PROGRAM Basic
VAR
	State:INT:= 0;
END_VAR

MC.Exec_Stop:= FALSE;
MC.Exec_Velocity := FALSE;

CASE state OF
	0:  MC.Exec_Stop:= TRUE;
		IF HMI.Bt_StartCycle THEN
			State:=1;
			MC.TargetDirection:= MC_Direction.MC_Positive_Direction;
			MC.TargetVel:= HMI.Tb_Vel;
		END_IF
	1:  MC.Exec_Velocity:=TRUE;
		IF HMI.Bt_StopCycle THEN
			State:=0;
		END_IF
END_CASE

END_PROGRAM

(* stored: Version 1.1.0.1, ProductVersion 3.1.4024.9
   POU Basic: Id {ce22bfcc-fbf0-4f66-8f8a-cc86cf734ace}, SpecialFunc None *)
